FUNCTION_BLOCK WithOutputs (* Only UPDATE updates the data inputs *)
  (* Standard: 61499-2; Description: Copyright (c) 2023 Johannes Kepler University Linz This program and the accompanying materials are made available under the terms of the Eclipse Public License 2.0 which is available at https://www.eclipse.org/legal/epl-2.0/ SPDX-License-Identifier: EPL-2.0 *)
  (* Version 1.0, 2023-03-07, Bianca Wiesmayr, Johannes Kepler University Linz, initial API and implementation and/or initial documentation *)
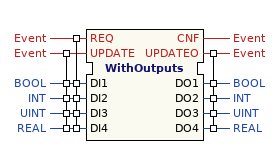
  EVENT_INPUT
    REQ WITH DI1, DI2, DI3, DI4;
    UPDATE WITH DI1, DI2, DI3, DI4;
  END_EVENT
  EVENT_OUTPUT
    CNF;
    UPDATEO WITH DO1, DO3, DO2, DO4;
  END_EVENT
  VAR_INPUT
    DI1 : BOOL;
    DI2 : INT;
    DI3 : UINT;
    DI4 : REAL;
  END_VAR
  VAR_OUTPUT
    DO1 : BOOL := 1;
    DO2 : INT := -42;
    DO3 : UINT := 21;
    DO4 : REAL := 3.14;
  END_VAR
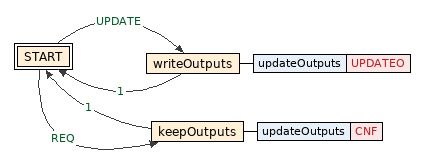
  EC_STATES
    START; (* Initial State *)
    writeOutputs : updateOutputs -> UPDATEO;
    keepOutputs : updateOutputs -> CNF;
  END_STATES
  EC_TRANSITIONS
    writeOutputs TO START := 1;
    START TO writeOutputs := UPDATE;
    START TO keepOutputs := REQ;
    keepOutputs TO START := 1;
  END_TRANSITIONS
  ALGORITHM updateOutputs IN ST:
DO1 := DI1;
DO2 := DI2;
DO3 := DI3;
DO4 := DI4;
  END_ALGORITHM
END_FUNCTION_BLOCK
